Omron CX-Programmer project NewProject (CX-Programmer 9.73)

# PLC NewPLC1: CP1E N20

## Global symbols (name address type ; comment)
0.01 BOOL  ; SENSOR
0.03 BOOL  ; RESET
100.03 BOOL  ; OUTPUT
C001 BOOL  ; COUNTER
C002 BOOL  ; COUNTER 2

## Program NewProgram1 (cyclic task 0)

### Section Section1

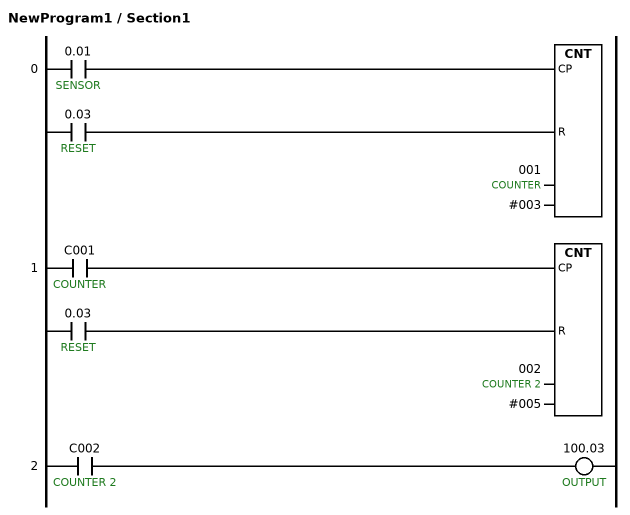
; rung 0
LD 0.01  ; SENSOR
LD 0.03  ; RESET
CNT 001 #003  ; COUNTER
; rung 1
LD C001  ; COUNTER
LD 0.03  ; RESET
CNT 002 #005  ; COUNTER 2
; rung 2
LD C002  ; COUNTER 2
OUT 100.03  ; OUTPUT

### Section END
; rung 0
END(001)